TYPE EM_Transport_Mechanische_Stop_ALM :
STRUCT
END_STRUCT
END_TYPE

(* stored: Version 1.1.0.1, ProductVersion 3.1.4024.12
   DUT EM_Transport_Mechanische_Stop_ALM: Id {a69b3629-6fe7-419f-9e27-88c0941a551d} *)
